Omron CX-Programmer project NewProject (CX-Programmer 9.73)

# PLC NewPLC1: CP1L M

## Global symbols (name address type ; comment)
0.00 BOOL  ; ACK
0.01 BOOL  ; RESET
0.02 BOOL  ; LAMP TEST
0.03 BOOL  ; LSH-D2017
0.04 BOOL  ; LSHH-D2017
0.05 BOOL  ; LSH-D2018
0.06 BOOL  ; LSHH-D2018
0.07 BOOL  ; LSH-O0001
0.08 BOOL  ; LSHH-O0001
0.09 BOOL  ; LSH-O0002
0.10 BOOL  ; LSHH-O0002
0.11 BOOL  ; LSH-O0003
100.00 BOOL  ; LAH-D2017
100.01 BOOL  ; LAHH-D2017
100.02 BOOL  ; LAH-D2018
100.03 BOOL  ; LAHH-D2018
100.04 BOOL  ; LAH-O0001
100.05 BOOL  ; LAHH-O0001
100.06 BOOL  ; LAH-O0002
100.07 BOOL  ; LAHH-O0002
101.00 BOOL  ; LAH-O0003
101.01 BOOL  ; LAHH-O0003
101.02 BOOL  ; LAH-O0004
101.03 BOOL  ; LAHH-O0004
101.04 BOOL  ; LAH-O0006
101.05 BOOL  ; LAHH-O0006
101.06 BOOL  ; LAH-O0008
101.07 BOOL  ; LAHH-O0008
102.00 BOOL  ; LAH-O0009
102.01 BOOL  ; LAHH-O0009
102.02 BOOL  ; LAH-O0010
102.03 BOOL  ; LAHH-O0010
102.04 BOOL  ; LAH-O0011
102.05 BOOL  ; LAHH-O0011
102.06 BOOL  ; LAH-O0012
102.07 BOOL  ; LAHH-O0012
103.00 BOOL  ; LAH-O0013
103.01 BOOL  ; LAHH-O0013
103.02 BOOL  ; LAH-O0014
103.03 BOOL  ; LAHH-O0014
103.04 BOOL  ; LAH-O0024
103.05 BOOL  ; LAHH-O0024
104.00 BOOL  ; LAH-O0025
104.01 BOOL  ; LAHH-O0025
104.02 BOOL  ; LAH-N0002
104.03 BOOL  ; LAHH-N0002
104.04 BOOL  ; LAH-N0004
104.05 BOOL  ; LAHH-N0004
104.06 BOOL  ; BUZZER
104.07 BOOL  ; HORN-LSH
105.00 BOOL  ; HORN-LSHH
105.01 BOOL  ; LIGHT-LSH
105.02 BOOL  ; LIGHT-LSHH
1.00 BOOL  ; LSHH-O0003
1.01 BOOL  ; LSH-O0004
1.02 BOOL  ; LSHH-O0004
1.03 BOOL  ; LSH-O0006
1.04 BOOL  ; LSHH-O0006
1.05 BOOL  ; LSH-O0008
1.06 BOOL  ; LSHH-O0008
2.00 BOOL  ; LSH-O0009
2.01 BOOL  ; LSHH-O0009
2.02 BOOL  ; LSH-O0010
2.03 BOOL  ; LSHH-O0010
2.04 BOOL  ; LSH-O0011
2.05 BOOL  ; LSHH-O0011
2.06 BOOL  ; LSH-O0012
2.07 BOOL  ; LSHH-O0012
2.08 BOOL  ; LSH-O0013
2.09 BOOL  ; LSHH-O0013
2.10 BOOL  ; LSH-O0014
2.11 BOOL  ; LSHH-O0014
3.00 BOOL  ; LSH-O0024
3.01 BOOL  ; LSHH-O0024
3.02 BOOL  ; LSH-O0025
3.03 BOOL  ; LSHH-O0025
3.04 BOOL  ; LSH-N0002
3.05 BOOL  ; LSHH-N0002
3.06 BOOL  ; LSH-N0004
3.07 BOOL  ; LSHH-N0004

## Program IHLAProject (cyclic task 0)

### Section RunningSystem

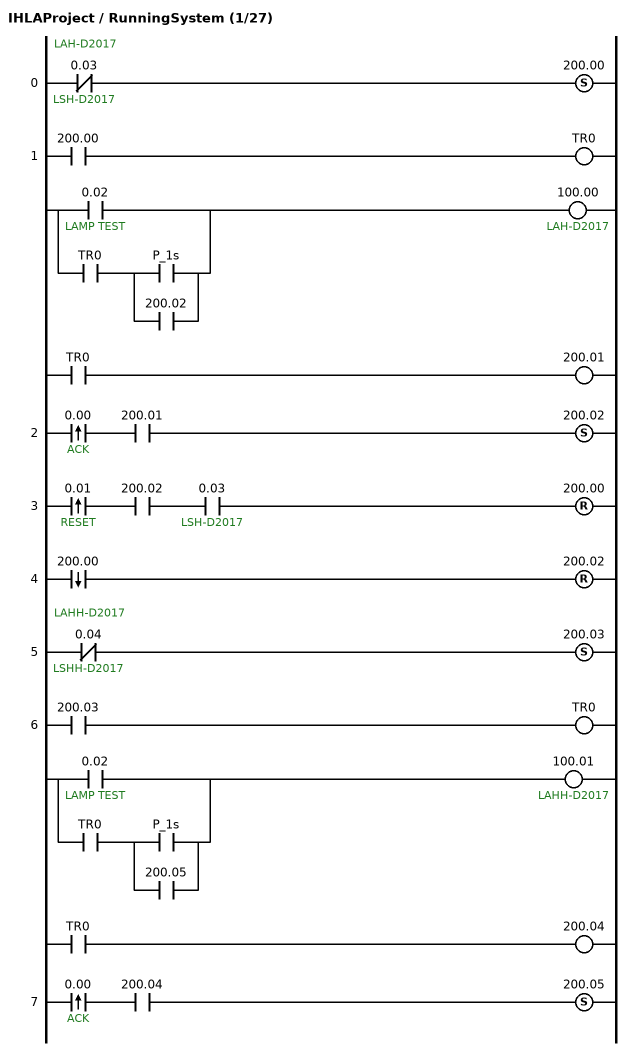
; rung 0: LAH-D2017
LDNOT 0.03  ; LSH-D2017
SET 200.00
; rung 1
LD 0.02  ; LAMP TEST
LD 200.00
OUT TR0
LD P_1s
OR 200.02
ANDLD
ORLD
OUT 100.00  ; LAH-D2017
LD TR0
OUT 200.01
; rung 2
@LD 0.00  ; ACK
AND 200.01
SET 200.02
; rung 3
@LD 0.01  ; RESET
AND 200.02
AND 0.03  ; LSH-D2017
RSET 200.00
; rung 4
%LD 200.00
RSET 200.02
; rung 5: LAHH-D2017
LDNOT 0.04  ; LSHH-D2017
SET 200.03
; rung 6
LD 0.02  ; LAMP TEST
LD 200.03
OUT TR0
LD P_1s
OR 200.05
ANDLD
ORLD
OUT 100.01  ; LAHH-D2017
LD TR0
OUT 200.04
; rung 7
@LD 0.00  ; ACK
AND 200.04
SET 200.05

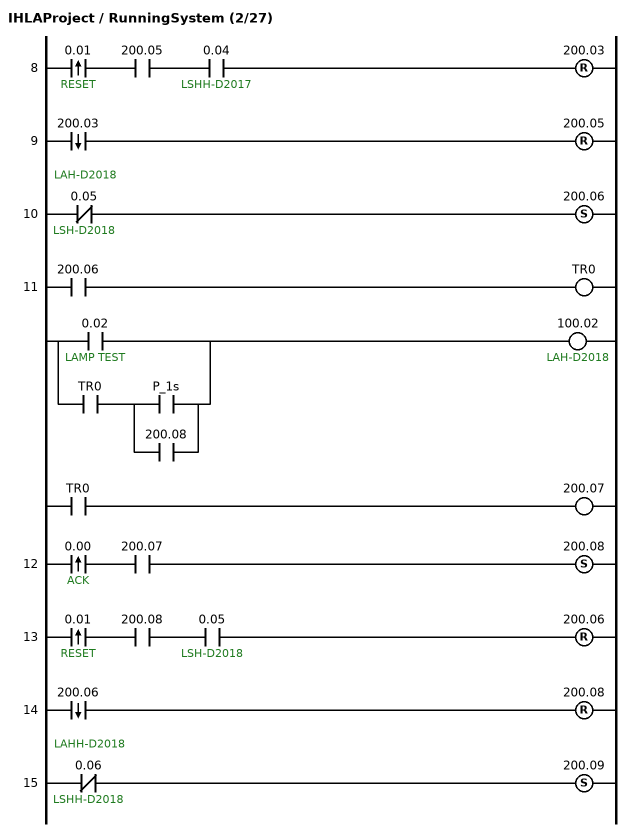
; rung 8
@LD 0.01  ; RESET
AND 200.05
AND 0.04  ; LSHH-D2017
RSET 200.03
; rung 9
%LD 200.03
RSET 200.05
; rung 10: LAH-D2018
LDNOT 0.05  ; LSH-D2018
SET 200.06
; rung 11
LD 0.02  ; LAMP TEST
LD 200.06
OUT TR0
LD P_1s
OR 200.08
ANDLD
ORLD
OUT 100.02  ; LAH-D2018
LD TR0
OUT 200.07
; rung 12
@LD 0.00  ; ACK
AND 200.07
SET 200.08
; rung 13
@LD 0.01  ; RESET
AND 200.08
AND 0.05  ; LSH-D2018
RSET 200.06
; rung 14
%LD 200.06
RSET 200.08
; rung 15: LAHH-D2018
LDNOT 0.06  ; LSHH-D2018
SET 200.09

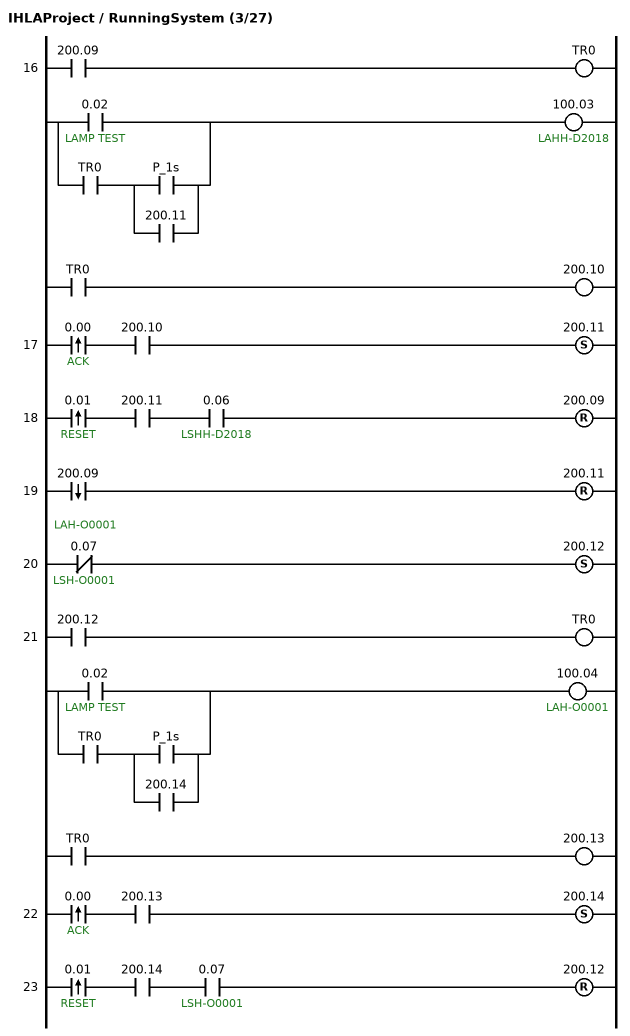
; rung 16
LD 0.02  ; LAMP TEST
LD 200.09
OUT TR0
LD P_1s
OR 200.11
ANDLD
ORLD
OUT 100.03  ; LAHH-D2018
LD TR0
OUT 200.10
; rung 17
@LD 0.00  ; ACK
AND 200.10
SET 200.11
; rung 18
@LD 0.01  ; RESET
AND 200.11
AND 0.06  ; LSHH-D2018
RSET 200.09
; rung 19
%LD 200.09
RSET 200.11
; rung 20: LAH-O0001
LDNOT 0.07  ; LSH-O0001
SET 200.12
; rung 21
LD 0.02  ; LAMP TEST
LD 200.12
OUT TR0
LD P_1s
OR 200.14
ANDLD
ORLD
OUT 100.04  ; LAH-O0001
LD TR0
OUT 200.13
; rung 22
@LD 0.00  ; ACK
AND 200.13
SET 200.14
; rung 23
@LD 0.01  ; RESET
AND 200.14
AND 0.07  ; LSH-O0001
RSET 200.12

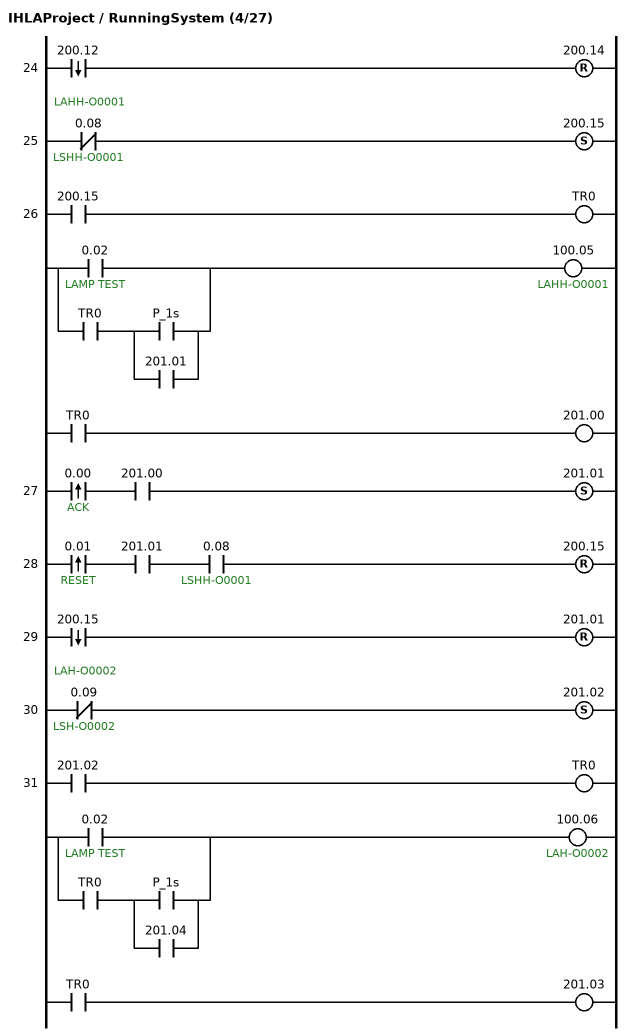
; rung 24
%LD 200.12
RSET 200.14
; rung 25: LAHH-O0001
LDNOT 0.08  ; LSHH-O0001
SET 200.15
; rung 26
LD 0.02  ; LAMP TEST
LD 200.15
OUT TR0
LD P_1s
OR 201.01
ANDLD
ORLD
OUT 100.05  ; LAHH-O0001
LD TR0
OUT 201.00
; rung 27
@LD 0.00  ; ACK
AND 201.00
SET 201.01
; rung 28
@LD 0.01  ; RESET
AND 201.01
AND 0.08  ; LSHH-O0001
RSET 200.15
; rung 29
%LD 200.15
RSET 201.01
; rung 30: LAH-O0002
LDNOT 0.09  ; LSH-O0002
SET 201.02
; rung 31
LD 0.02  ; LAMP TEST
LD 201.02
OUT TR0
LD P_1s
OR 201.04
ANDLD
ORLD
OUT 100.06  ; LAH-O0002
LD TR0
OUT 201.03

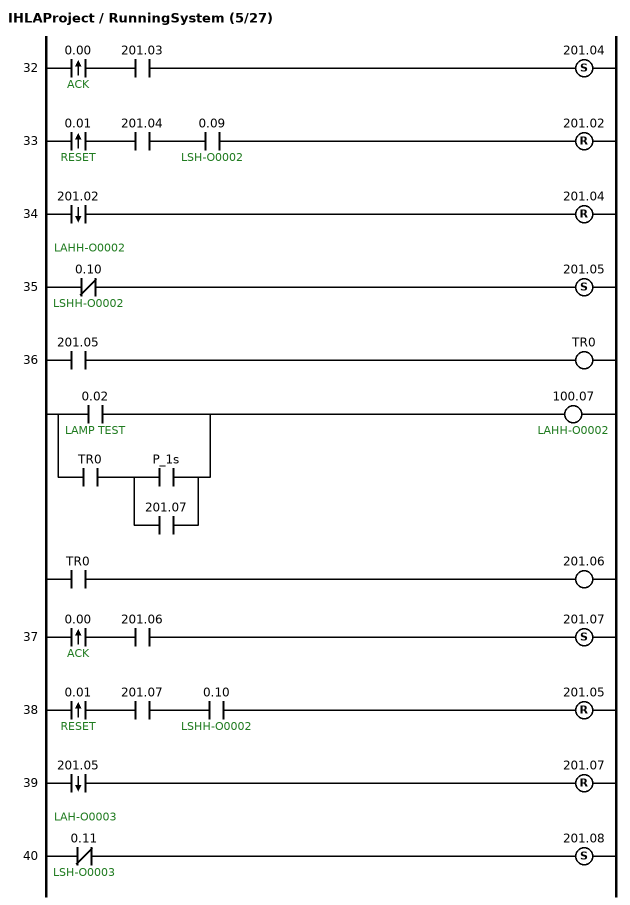
; rung 32
@LD 0.00  ; ACK
AND 201.03
SET 201.04
; rung 33
@LD 0.01  ; RESET
AND 201.04
AND 0.09  ; LSH-O0002
RSET 201.02
; rung 34
%LD 201.02
RSET 201.04
; rung 35: LAHH-O0002
LDNOT 0.10  ; LSHH-O0002
SET 201.05
; rung 36
LD 0.02  ; LAMP TEST
LD 201.05
OUT TR0
LD P_1s
OR 201.07
ANDLD
ORLD
OUT 100.07  ; LAHH-O0002
LD TR0
OUT 201.06
; rung 37
@LD 0.00  ; ACK
AND 201.06
SET 201.07
; rung 38
@LD 0.01  ; RESET
AND 201.07
AND 0.10  ; LSHH-O0002
RSET 201.05
; rung 39
%LD 201.05
RSET 201.07
; rung 40: LAH-O0003
LDNOT 0.11  ; LSH-O0003
SET 201.08

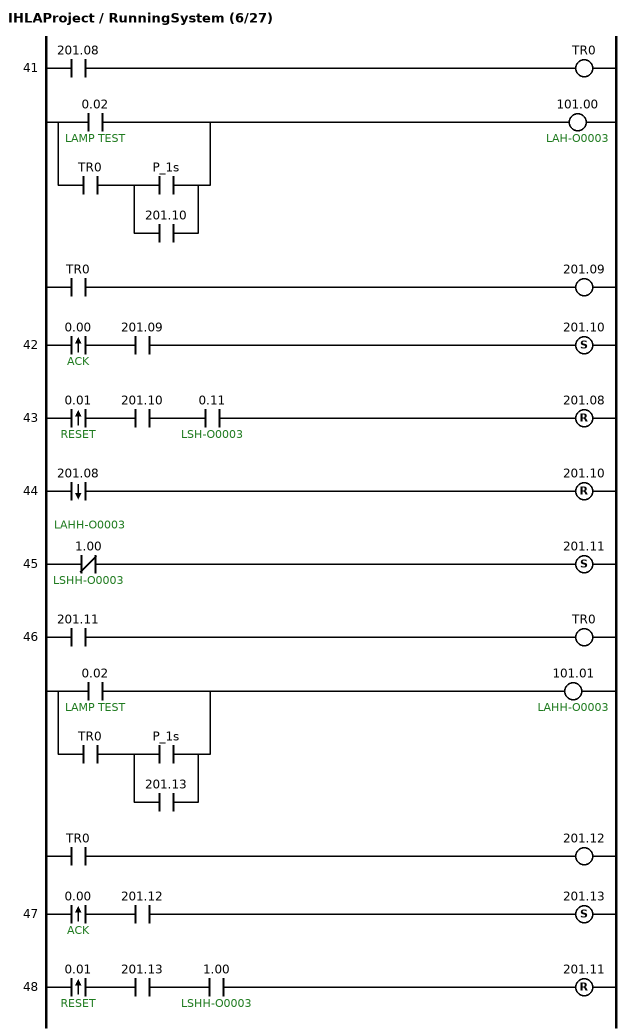
; rung 41
LD 0.02  ; LAMP TEST
LD 201.08
OUT TR0
LD P_1s
OR 201.10
ANDLD
ORLD
OUT 101.00  ; LAH-O0003
LD TR0
OUT 201.09
; rung 42
@LD 0.00  ; ACK
AND 201.09
SET 201.10
; rung 43
@LD 0.01  ; RESET
AND 201.10
AND 0.11  ; LSH-O0003
RSET 201.08
; rung 44
%LD 201.08
RSET 201.10
; rung 45: LAHH-O0003
LDNOT 1.00  ; LSHH-O0003
SET 201.11
; rung 46
LD 0.02  ; LAMP TEST
LD 201.11
OUT TR0
LD P_1s
OR 201.13
ANDLD
ORLD
OUT 101.01  ; LAHH-O0003
LD TR0
OUT 201.12
; rung 47
@LD 0.00  ; ACK
AND 201.12
SET 201.13
; rung 48
@LD 0.01  ; RESET
AND 201.13
AND 1.00  ; LSHH-O0003
RSET 201.11

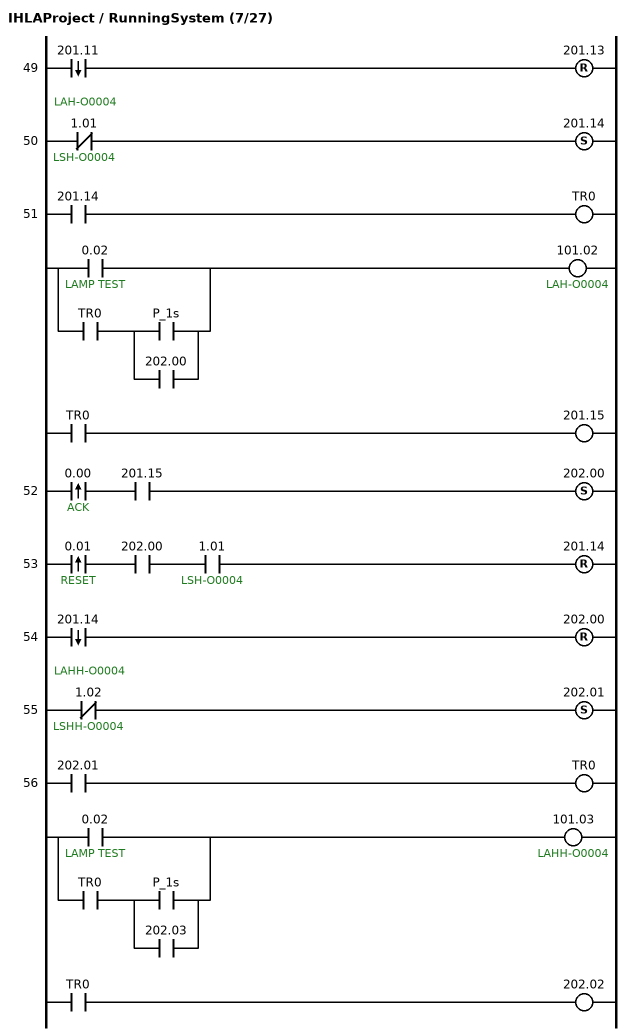
; rung 49
%LD 201.11
RSET 201.13
; rung 50: LAH-O0004
LDNOT 1.01  ; LSH-O0004
SET 201.14
; rung 51
LD 0.02  ; LAMP TEST
LD 201.14
OUT TR0
LD P_1s
OR 202.00
ANDLD
ORLD
OUT 101.02  ; LAH-O0004
LD TR0
OUT 201.15
; rung 52
@LD 0.00  ; ACK
AND 201.15
SET 202.00
; rung 53
@LD 0.01  ; RESET
AND 202.00
AND 1.01  ; LSH-O0004
RSET 201.14
; rung 54
%LD 201.14
RSET 202.00
; rung 55: LAHH-O0004
LDNOT 1.02  ; LSHH-O0004
SET 202.01
; rung 56
LD 0.02  ; LAMP TEST
LD 202.01
OUT TR0
LD P_1s
OR 202.03
ANDLD
ORLD
OUT 101.03  ; LAHH-O0004
LD TR0
OUT 202.02

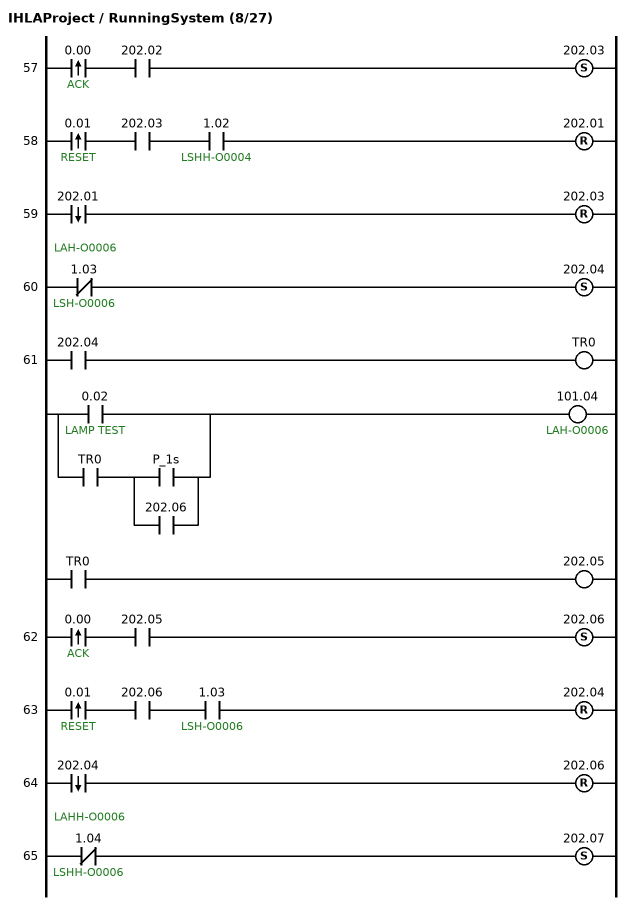
; rung 57
@LD 0.00  ; ACK
AND 202.02
SET 202.03
; rung 58
@LD 0.01  ; RESET
AND 202.03
AND 1.02  ; LSHH-O0004
RSET 202.01
; rung 59
%LD 202.01
RSET 202.03
; rung 60: LAH-O0006
LDNOT 1.03  ; LSH-O0006
SET 202.04
; rung 61
LD 0.02  ; LAMP TEST
LD 202.04
OUT TR0
LD P_1s
OR 202.06
ANDLD
ORLD
OUT 101.04  ; LAH-O0006
LD TR0
OUT 202.05
; rung 62
@LD 0.00  ; ACK
AND 202.05
SET 202.06
; rung 63
@LD 0.01  ; RESET
AND 202.06
AND 1.03  ; LSH-O0006
RSET 202.04
; rung 64
%LD 202.04
RSET 202.06
; rung 65: LAHH-O0006
LDNOT 1.04  ; LSHH-O0006
SET 202.07

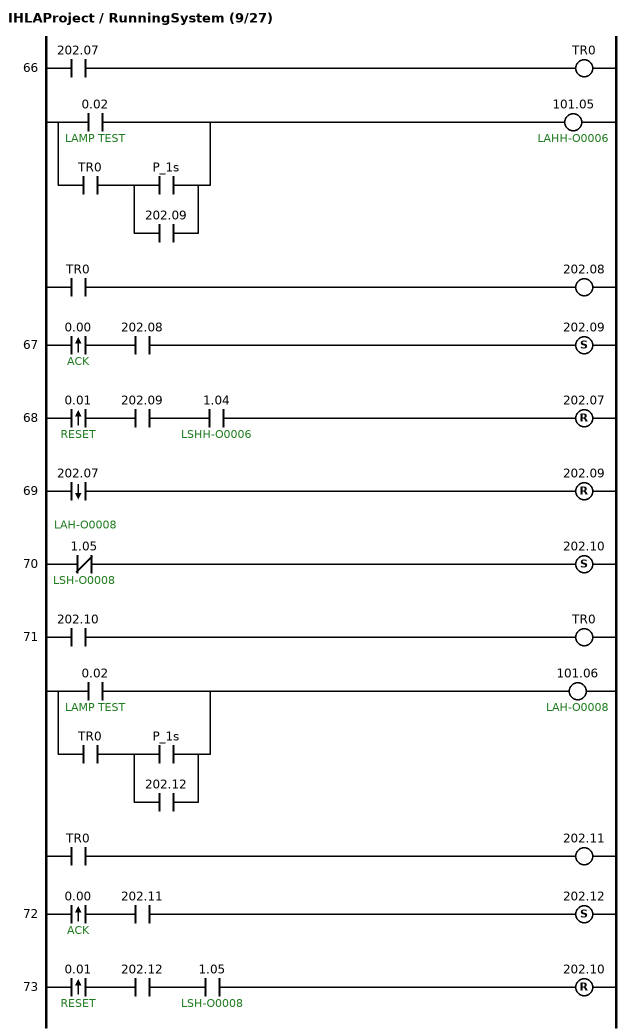
; rung 66
LD 0.02  ; LAMP TEST
LD 202.07
OUT TR0
LD P_1s
OR 202.09
ANDLD
ORLD
OUT 101.05  ; LAHH-O0006
LD TR0
OUT 202.08
; rung 67
@LD 0.00  ; ACK
AND 202.08
SET 202.09
; rung 68
@LD 0.01  ; RESET
AND 202.09
AND 1.04  ; LSHH-O0006
RSET 202.07
; rung 69
%LD 202.07
RSET 202.09
; rung 70: LAH-O0008
LDNOT 1.05  ; LSH-O0008
SET 202.10
; rung 71
LD 0.02  ; LAMP TEST
LD 202.10
OUT TR0
LD P_1s
OR 202.12
ANDLD
ORLD
OUT 101.06  ; LAH-O0008
LD TR0
OUT 202.11
; rung 72
@LD 0.00  ; ACK
AND 202.11
SET 202.12
; rung 73
@LD 0.01  ; RESET
AND 202.12
AND 1.05  ; LSH-O0008
RSET 202.10

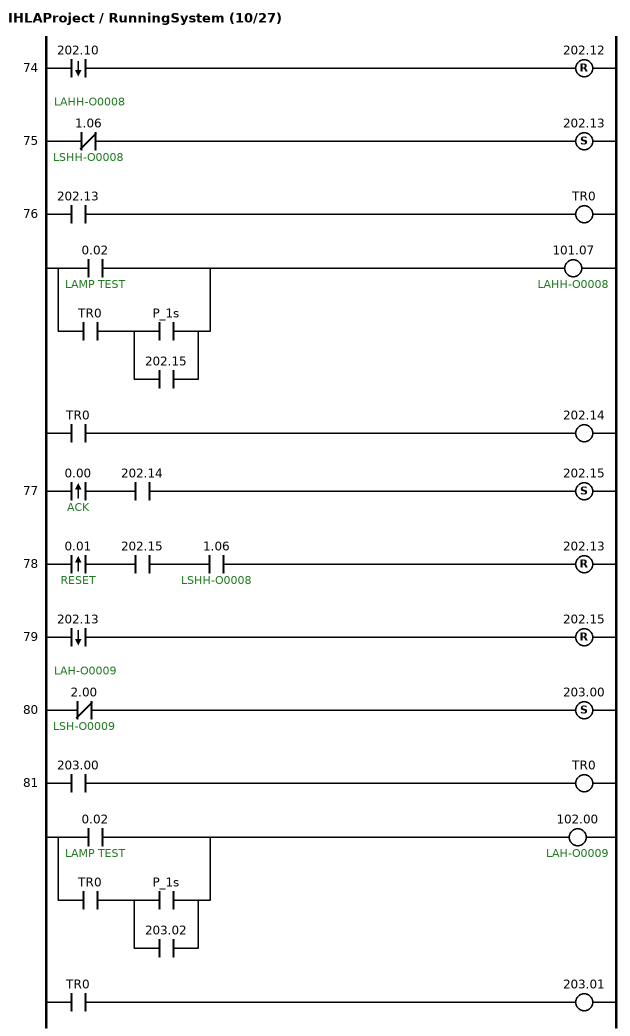
; rung 74
%LD 202.10
RSET 202.12
; rung 75: LAHH-O0008
LDNOT 1.06  ; LSHH-O0008
SET 202.13
; rung 76
LD 0.02  ; LAMP TEST
LD 202.13
OUT TR0
LD P_1s
OR 202.15
ANDLD
ORLD
OUT 101.07  ; LAHH-O0008
LD TR0
OUT 202.14
; rung 77
@LD 0.00  ; ACK
AND 202.14
SET 202.15
; rung 78
@LD 0.01  ; RESET
AND 202.15
AND 1.06  ; LSHH-O0008
RSET 202.13
; rung 79
%LD 202.13
RSET 202.15
; rung 80: LAH-O0009
LDNOT 2.00  ; LSH-O0009
SET 203.00
; rung 81
LD 0.02  ; LAMP TEST
LD 203.00
OUT TR0
LD P_1s
OR 203.02
ANDLD
ORLD
OUT 102.00  ; LAH-O0009
LD TR0
OUT 203.01

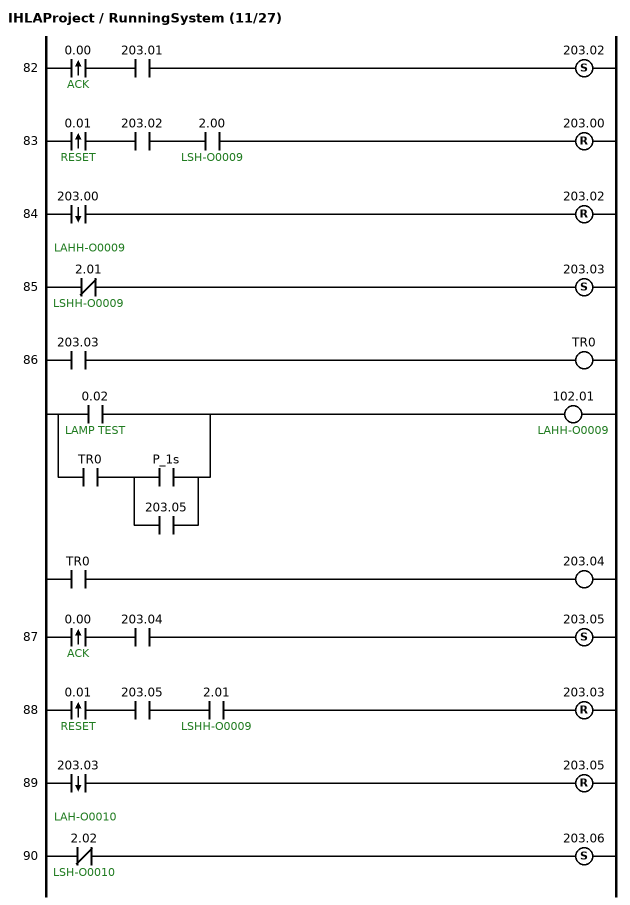
; rung 82
@LD 0.00  ; ACK
AND 203.01
SET 203.02
; rung 83
@LD 0.01  ; RESET
AND 203.02
AND 2.00  ; LSH-O0009
RSET 203.00
; rung 84
%LD 203.00
RSET 203.02
; rung 85: LAHH-O0009
LDNOT 2.01  ; LSHH-O0009
SET 203.03
; rung 86
LD 0.02  ; LAMP TEST
LD 203.03
OUT TR0
LD P_1s
OR 203.05
ANDLD
ORLD
OUT 102.01  ; LAHH-O0009
LD TR0
OUT 203.04
; rung 87
@LD 0.00  ; ACK
AND 203.04
SET 203.05
; rung 88
@LD 0.01  ; RESET
AND 203.05
AND 2.01  ; LSHH-O0009
RSET 203.03
; rung 89
%LD 203.03
RSET 203.05
; rung 90: LAH-O0010
LDNOT 2.02  ; LSH-O0010
SET 203.06

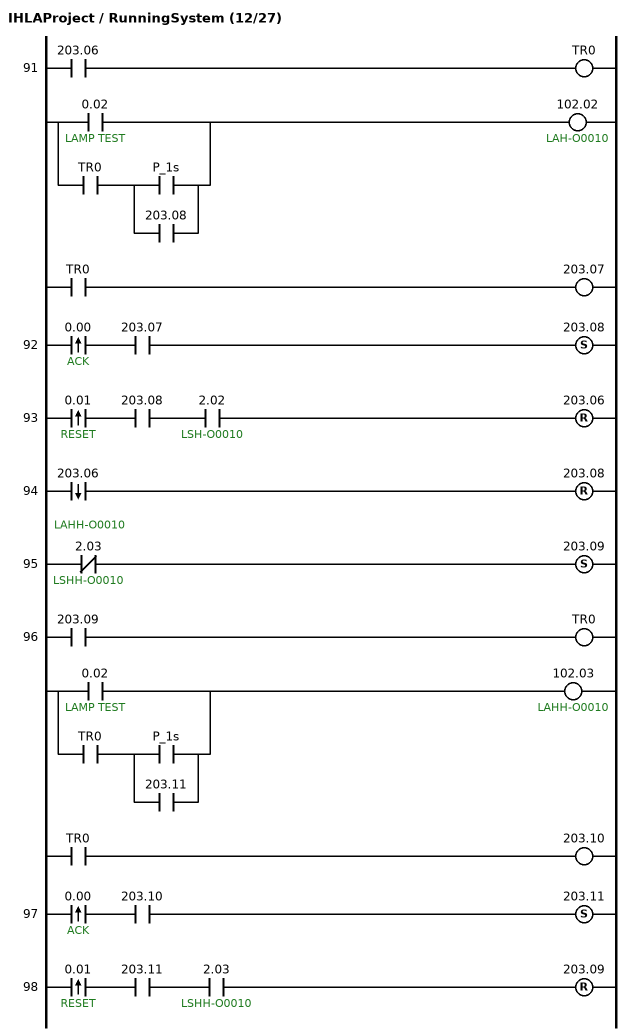
; rung 91
LD 0.02  ; LAMP TEST
LD 203.06
OUT TR0
LD P_1s
OR 203.08
ANDLD
ORLD
OUT 102.02  ; LAH-O0010
LD TR0
OUT 203.07
; rung 92
@LD 0.00  ; ACK
AND 203.07
SET 203.08
; rung 93
@LD 0.01  ; RESET
AND 203.08
AND 2.02  ; LSH-O0010
RSET 203.06
; rung 94
%LD 203.06
RSET 203.08
; rung 95: LAHH-O0010
LDNOT 2.03  ; LSHH-O0010
SET 203.09
; rung 96
LD 0.02  ; LAMP TEST
LD 203.09
OUT TR0
LD P_1s
OR 203.11
ANDLD
ORLD
OUT 102.03  ; LAHH-O0010
LD TR0
OUT 203.10
; rung 97
@LD 0.00  ; ACK
AND 203.10
SET 203.11
; rung 98
@LD 0.01  ; RESET
AND 203.11
AND 2.03  ; LSHH-O0010
RSET 203.09

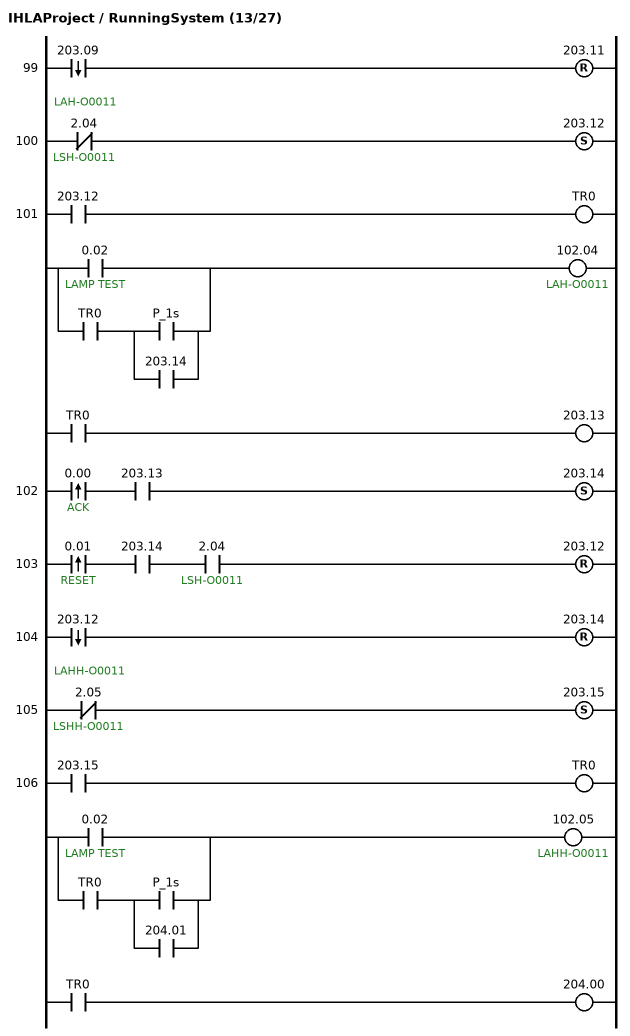
; rung 99
%LD 203.09
RSET 203.11
; rung 100: LAH-O0011
LDNOT 2.04  ; LSH-O0011
SET 203.12
; rung 101
LD 0.02  ; LAMP TEST
LD 203.12
OUT TR0
LD P_1s
OR 203.14
ANDLD
ORLD
OUT 102.04  ; LAH-O0011
LD TR0
OUT 203.13
; rung 102
@LD 0.00  ; ACK
AND 203.13
SET 203.14
; rung 103
@LD 0.01  ; RESET
AND 203.14
AND 2.04  ; LSH-O0011
RSET 203.12
; rung 104
%LD 203.12
RSET 203.14
; rung 105: LAHH-O0011
LDNOT 2.05  ; LSHH-O0011
SET 203.15
; rung 106
LD 0.02  ; LAMP TEST
LD 203.15
OUT TR0
LD P_1s
OR 204.01
ANDLD
ORLD
OUT 102.05  ; LAHH-O0011
LD TR0
OUT 204.00

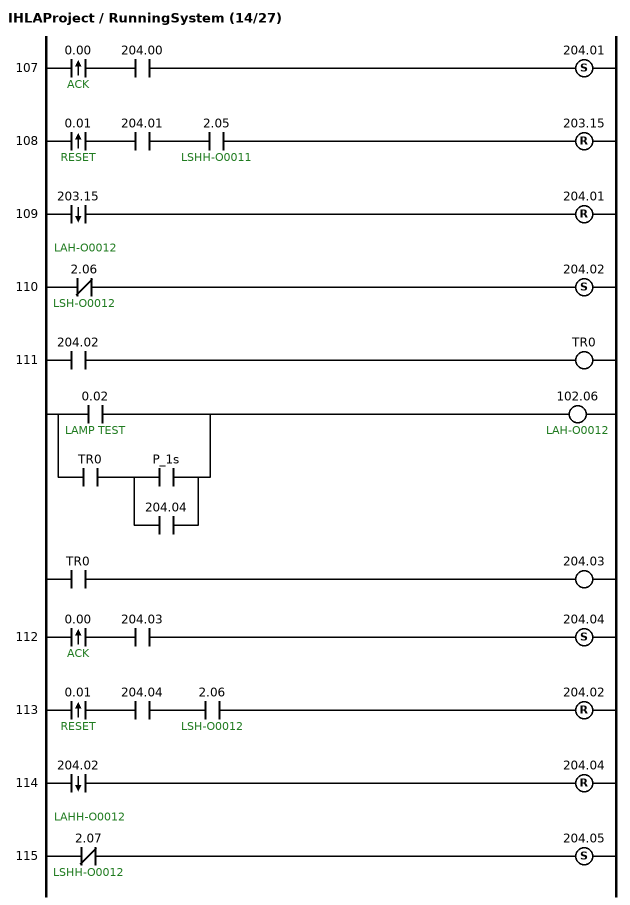
; rung 107
@LD 0.00  ; ACK
AND 204.00
SET 204.01
; rung 108
@LD 0.01  ; RESET
AND 204.01
AND 2.05  ; LSHH-O0011
RSET 203.15
; rung 109
%LD 203.15
RSET 204.01
; rung 110: LAH-O0012
LDNOT 2.06  ; LSH-O0012
SET 204.02
; rung 111
LD 0.02  ; LAMP TEST
LD 204.02
OUT TR0
LD P_1s
OR 204.04
ANDLD
ORLD
OUT 102.06  ; LAH-O0012
LD TR0
OUT 204.03
; rung 112
@LD 0.00  ; ACK
AND 204.03
SET 204.04
; rung 113
@LD 0.01  ; RESET
AND 204.04
AND 2.06  ; LSH-O0012
RSET 204.02
; rung 114
%LD 204.02
RSET 204.04
; rung 115: LAHH-O0012
LDNOT 2.07  ; LSHH-O0012
SET 204.05

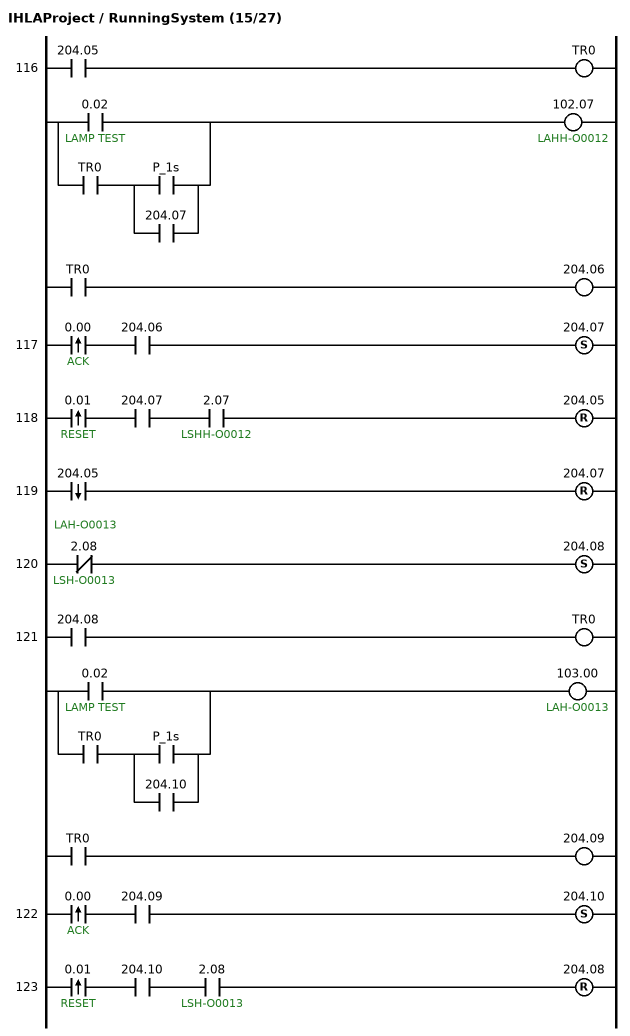
; rung 116
LD 0.02  ; LAMP TEST
LD 204.05
OUT TR0
LD P_1s
OR 204.07
ANDLD
ORLD
OUT 102.07  ; LAHH-O0012
LD TR0
OUT 204.06
; rung 117
@LD 0.00  ; ACK
AND 204.06
SET 204.07
; rung 118
@LD 0.01  ; RESET
AND 204.07
AND 2.07  ; LSHH-O0012
RSET 204.05
; rung 119
%LD 204.05
RSET 204.07
; rung 120: LAH-O0013
LDNOT 2.08  ; LSH-O0013
SET 204.08
; rung 121
LD 0.02  ; LAMP TEST
LD 204.08
OUT TR0
LD P_1s
OR 204.10
ANDLD
ORLD
OUT 103.00  ; LAH-O0013
LD TR0
OUT 204.09
; rung 122
@LD 0.00  ; ACK
AND 204.09
SET 204.10
; rung 123
@LD 0.01  ; RESET
AND 204.10
AND 2.08  ; LSH-O0013
RSET 204.08

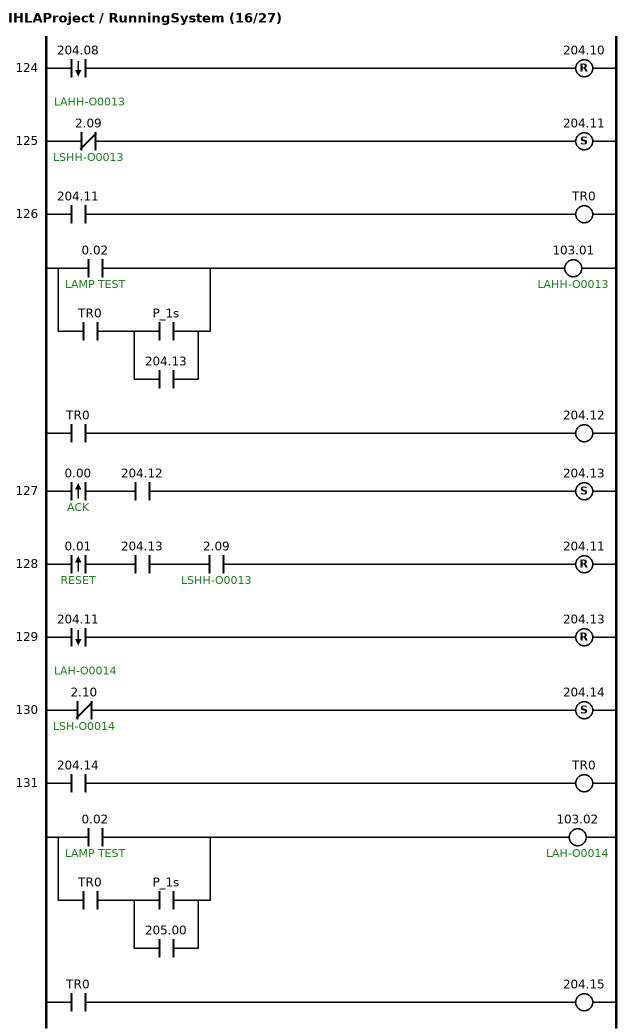
; rung 124
%LD 204.08
RSET 204.10
; rung 125: LAHH-O0013
LDNOT 2.09  ; LSHH-O0013
SET 204.11
; rung 126
LD 0.02  ; LAMP TEST
LD 204.11
OUT TR0
LD P_1s
OR 204.13
ANDLD
ORLD
OUT 103.01  ; LAHH-O0013
LD TR0
OUT 204.12
; rung 127
@LD 0.00  ; ACK
AND 204.12
SET 204.13
; rung 128
@LD 0.01  ; RESET
AND 204.13
AND 2.09  ; LSHH-O0013
RSET 204.11
; rung 129
%LD 204.11
RSET 204.13
; rung 130: LAH-O0014
LDNOT 2.10  ; LSH-O0014
SET 204.14
; rung 131
LD 0.02  ; LAMP TEST
LD 204.14
OUT TR0
LD P_1s
OR 205.00
ANDLD
ORLD
OUT 103.02  ; LAH-O0014
LD TR0
OUT 204.15

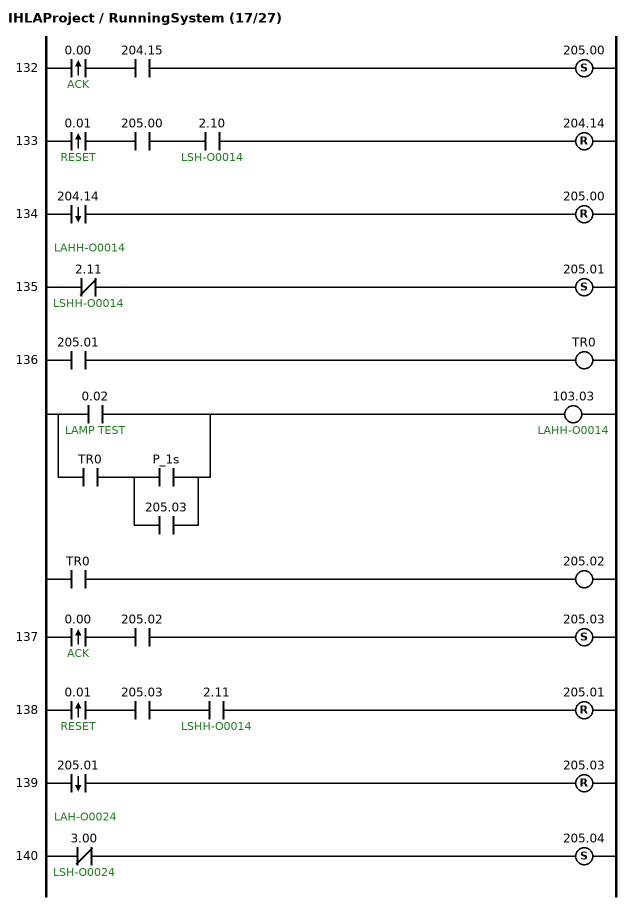
; rung 132
@LD 0.00  ; ACK
AND 204.15
SET 205.00
; rung 133
@LD 0.01  ; RESET
AND 205.00
AND 2.10  ; LSH-O0014
RSET 204.14
; rung 134
%LD 204.14
RSET 205.00
; rung 135: LAHH-O0014
LDNOT 2.11  ; LSHH-O0014
SET 205.01
; rung 136
LD 0.02  ; LAMP TEST
LD 205.01
OUT TR0
LD P_1s
OR 205.03
ANDLD
ORLD
OUT 103.03  ; LAHH-O0014
LD TR0
OUT 205.02
; rung 137
@LD 0.00  ; ACK
AND 205.02
SET 205.03
; rung 138
@LD 0.01  ; RESET
AND 205.03
AND 2.11  ; LSHH-O0014
RSET 205.01
; rung 139
%LD 205.01
RSET 205.03
; rung 140: LAH-O0024
LDNOT 3.00  ; LSH-O0024
SET 205.04

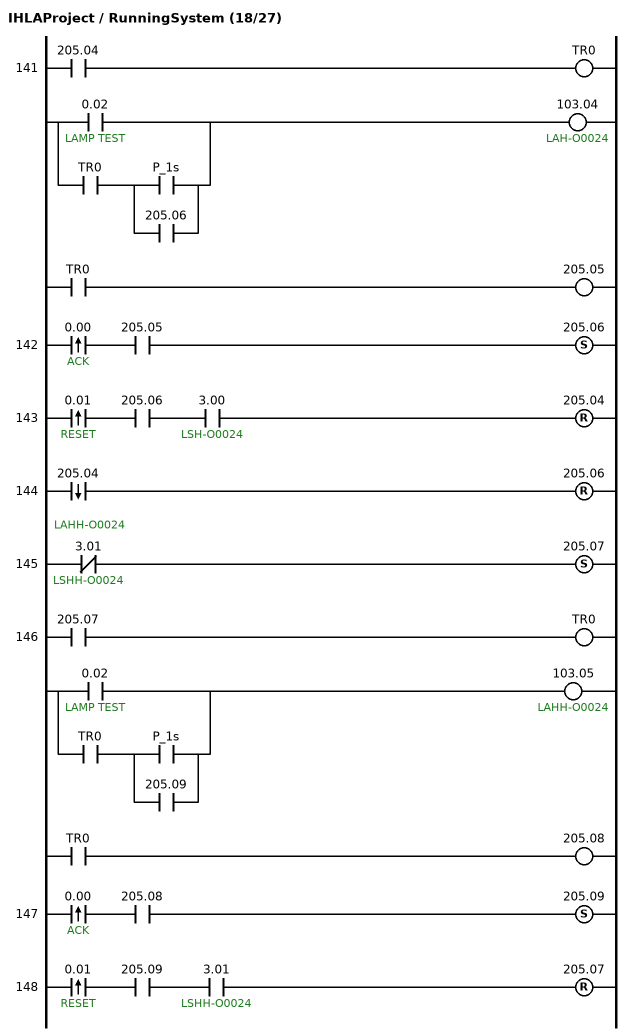
; rung 141
LD 0.02  ; LAMP TEST
LD 205.04
OUT TR0
LD P_1s
OR 205.06
ANDLD
ORLD
OUT 103.04  ; LAH-O0024
LD TR0
OUT 205.05
; rung 142
@LD 0.00  ; ACK
AND 205.05
SET 205.06
; rung 143
@LD 0.01  ; RESET
AND 205.06
AND 3.00  ; LSH-O0024
RSET 205.04
; rung 144
%LD 205.04
RSET 205.06
; rung 145: LAHH-O0024
LDNOT 3.01  ; LSHH-O0024
SET 205.07
; rung 146
LD 0.02  ; LAMP TEST
LD 205.07
OUT TR0
LD P_1s
OR 205.09
ANDLD
ORLD
OUT 103.05  ; LAHH-O0024
LD TR0
OUT 205.08
; rung 147
@LD 0.00  ; ACK
AND 205.08
SET 205.09
; rung 148
@LD 0.01  ; RESET
AND 205.09
AND 3.01  ; LSHH-O0024
RSET 205.07

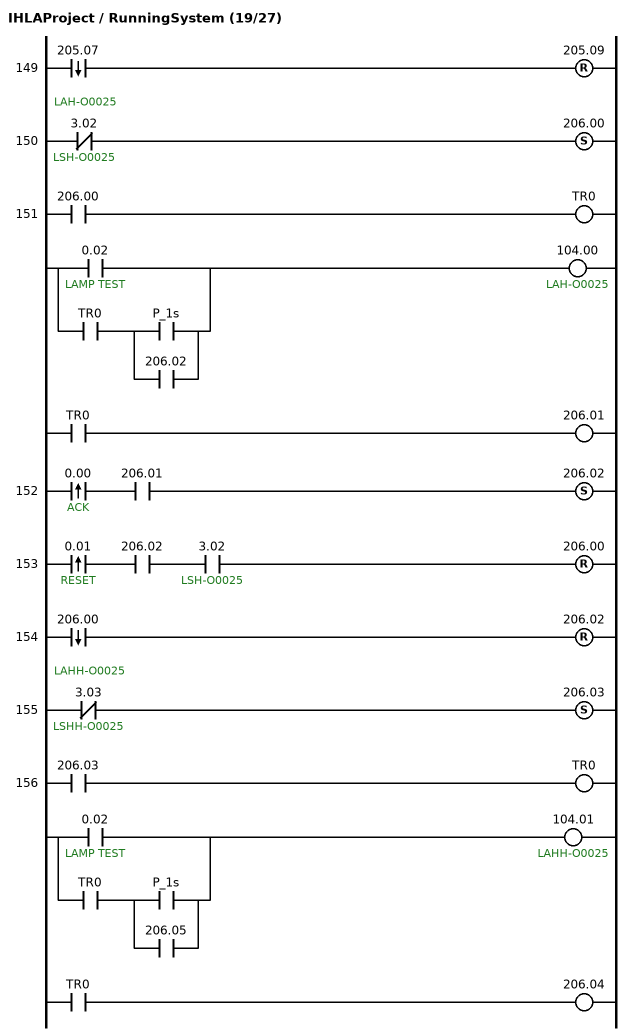
; rung 149
%LD 205.07
RSET 205.09
; rung 150: LAH-O0025
LDNOT 3.02  ; LSH-O0025
SET 206.00
; rung 151
LD 0.02  ; LAMP TEST
LD 206.00
OUT TR0
LD P_1s
OR 206.02
ANDLD
ORLD
OUT 104.00  ; LAH-O0025
LD TR0
OUT 206.01
; rung 152
@LD 0.00  ; ACK
AND 206.01
SET 206.02
; rung 153
@LD 0.01  ; RESET
AND 206.02
AND 3.02  ; LSH-O0025
RSET 206.00
; rung 154
%LD 206.00
RSET 206.02
; rung 155: LAHH-O0025
LDNOT 3.03  ; LSHH-O0025
SET 206.03
; rung 156
LD 0.02  ; LAMP TEST
LD 206.03
OUT TR0
LD P_1s
OR 206.05
ANDLD
ORLD
OUT 104.01  ; LAHH-O0025
LD TR0
OUT 206.04

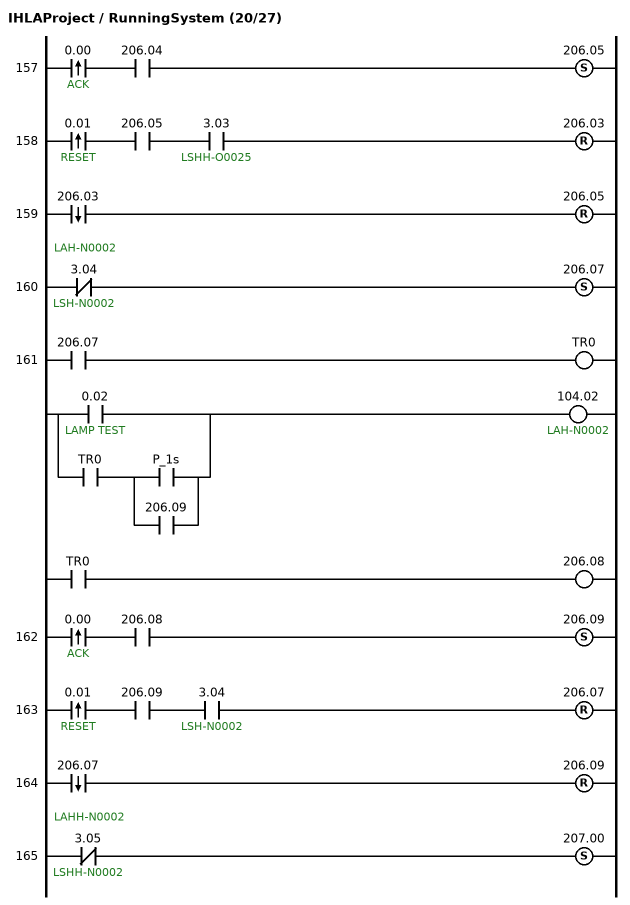
; rung 157
@LD 0.00  ; ACK
AND 206.04
SET 206.05
; rung 158
@LD 0.01  ; RESET
AND 206.05
AND 3.03  ; LSHH-O0025
RSET 206.03
; rung 159
%LD 206.03
RSET 206.05
; rung 160: LAH-N0002
LDNOT 3.04  ; LSH-N0002
SET 206.07
; rung 161
LD 0.02  ; LAMP TEST
LD 206.07
OUT TR0
LD P_1s
OR 206.09
ANDLD
ORLD
OUT 104.02  ; LAH-N0002
LD TR0
OUT 206.08
; rung 162
@LD 0.00  ; ACK
AND 206.08
SET 206.09
; rung 163
@LD 0.01  ; RESET
AND 206.09
AND 3.04  ; LSH-N0002
RSET 206.07
; rung 164
%LD 206.07
RSET 206.09
; rung 165: LAHH-N0002
LDNOT 3.05  ; LSHH-N0002
SET 207.00

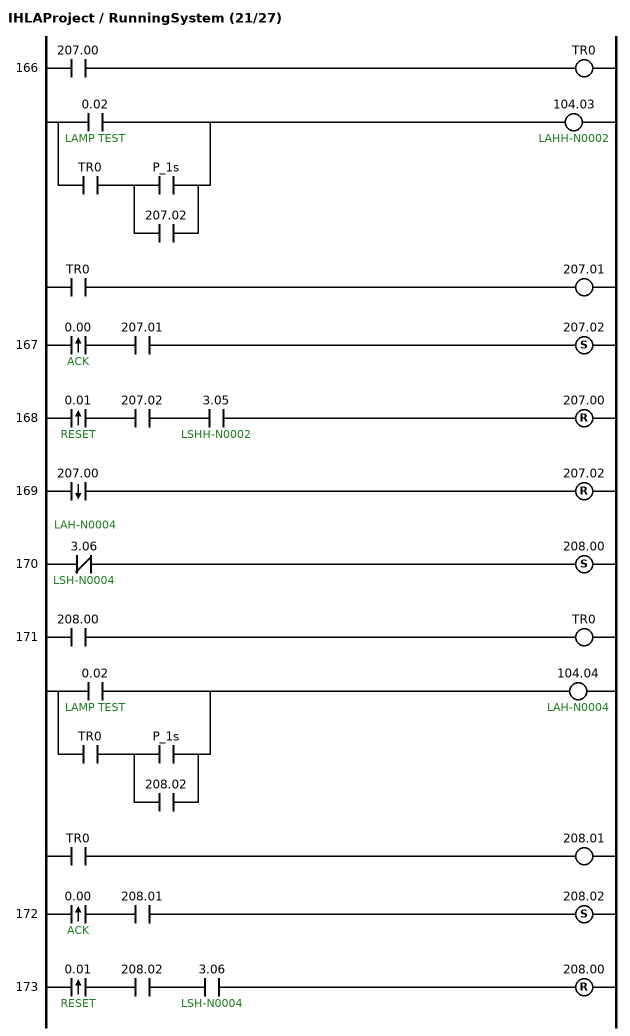
; rung 166
LD 0.02  ; LAMP TEST
LD 207.00
OUT TR0
LD P_1s
OR 207.02
ANDLD
ORLD
OUT 104.03  ; LAHH-N0002
LD TR0
OUT 207.01
; rung 167
@LD 0.00  ; ACK
AND 207.01
SET 207.02
; rung 168
@LD 0.01  ; RESET
AND 207.02
AND 3.05  ; LSHH-N0002
RSET 207.00
; rung 169
%LD 207.00
RSET 207.02
; rung 170: LAH-N0004
LDNOT 3.06  ; LSH-N0004
SET 208.00
; rung 171
LD 0.02  ; LAMP TEST
LD 208.00
OUT TR0
LD P_1s
OR 208.02
ANDLD
ORLD
OUT 104.04  ; LAH-N0004
LD TR0
OUT 208.01
; rung 172
@LD 0.00  ; ACK
AND 208.01
SET 208.02
; rung 173
@LD 0.01  ; RESET
AND 208.02
AND 3.06  ; LSH-N0004
RSET 208.00

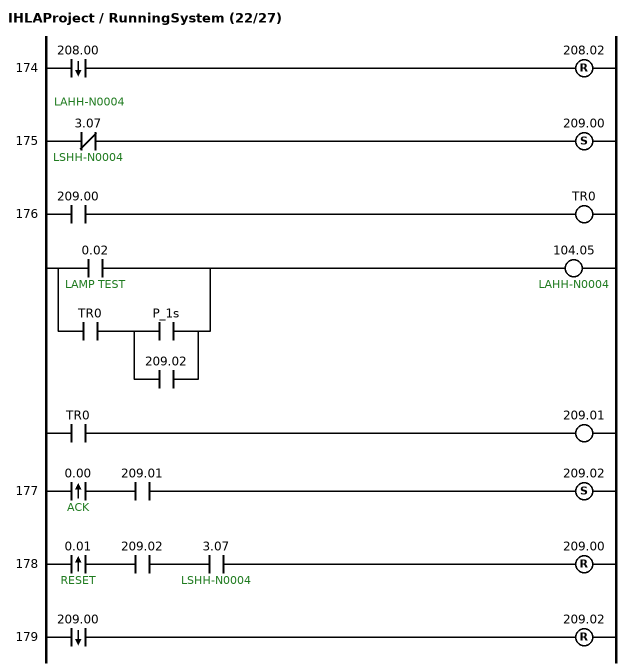
; rung 174
%LD 208.00
RSET 208.02
; rung 175: LAHH-N0004
LDNOT 3.07  ; LSHH-N0004
SET 209.00
; rung 176
LD 0.02  ; LAMP TEST
LD 209.00
OUT TR0
LD P_1s
OR 209.02
ANDLD
ORLD
OUT 104.05  ; LAHH-N0004
LD TR0
OUT 209.01
; rung 177
@LD 0.00  ; ACK
AND 209.01
SET 209.02
; rung 178
@LD 0.01  ; RESET
AND 209.02
AND 3.07  ; LSHH-N0004
RSET 209.00
; rung 179
%LD 209.00
RSET 209.02

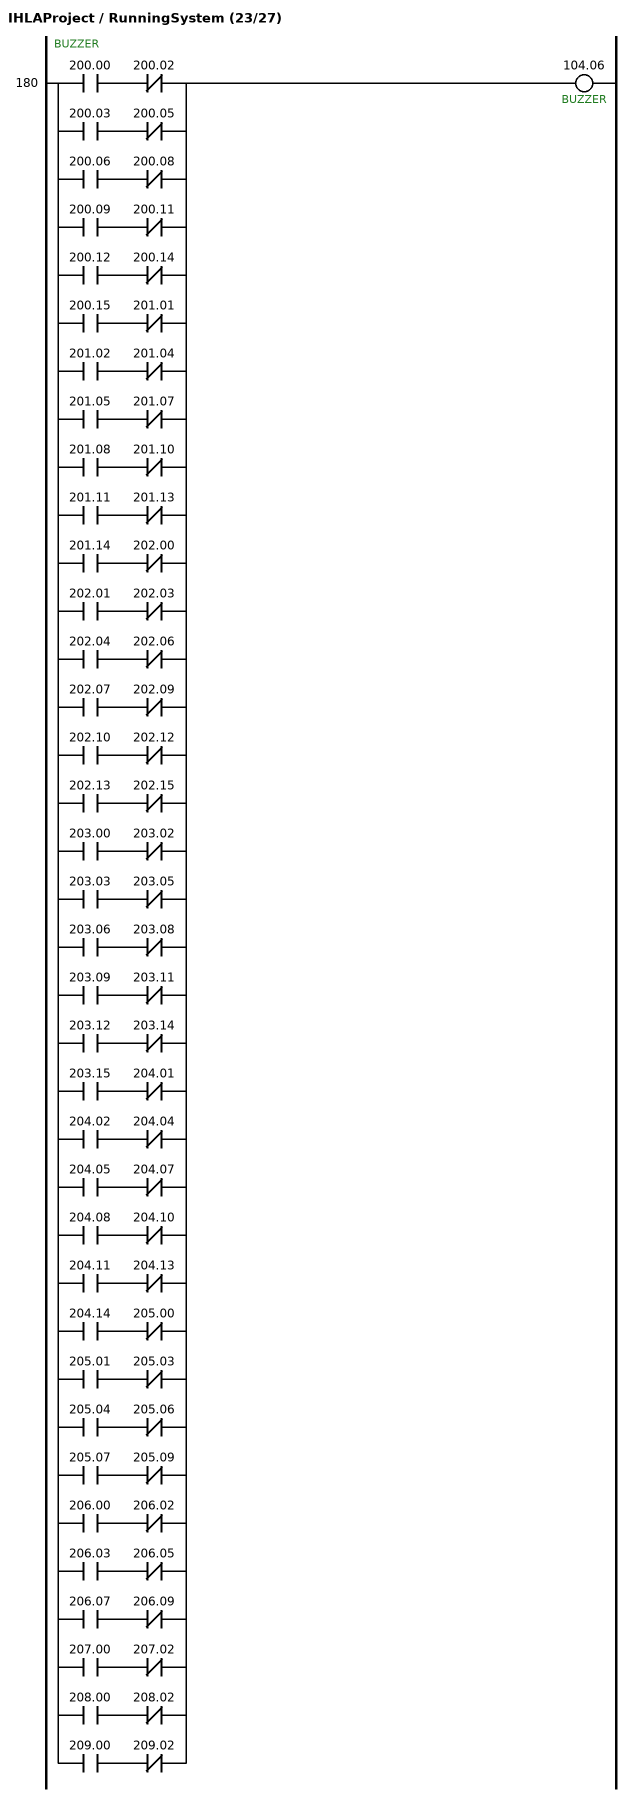
; rung 180: BUZZER
LD 200.00
ANDNOT 200.02
LD 200.03
ANDNOT 200.05
ORLD
LD 200.06
ANDNOT 200.08
ORLD
LD 200.09
ANDNOT 200.11
ORLD
LD 200.12
ANDNOT 200.14
ORLD
LD 200.15
ANDNOT 201.01
ORLD
LD 201.02
ANDNOT 201.04
ORLD
LD 201.05
ANDNOT 201.07
ORLD
LD 201.08
ANDNOT 201.10
ORLD
LD 201.11
ANDNOT 201.13
ORLD
LD 201.14
ANDNOT 202.00
ORLD
LD 202.01
ANDNOT 202.03
ORLD
LD 202.04
ANDNOT 202.06
ORLD
LD 202.07
ANDNOT 202.09
ORLD
LD 202.10
ANDNOT 202.12
ORLD
LD 202.13
ANDNOT 202.15
ORLD
LD 203.00
ANDNOT 203.02
ORLD
LD 203.03
ANDNOT 203.05
ORLD
LD 203.06
ANDNOT 203.08
ORLD
LD 203.09
ANDNOT 203.11
ORLD
LD 203.12
ANDNOT 203.14
ORLD
LD 203.15
ANDNOT 204.01
ORLD
LD 204.02
ANDNOT 204.04
ORLD
LD 204.05
ANDNOT 204.07
ORLD
LD 204.08
ANDNOT 204.10
ORLD
LD 204.11
ANDNOT 204.13
ORLD
LD 204.14
ANDNOT 205.00
ORLD
LD 205.01
ANDNOT 205.03
ORLD
LD 205.04
ANDNOT 205.06
ORLD
LD 205.07
ANDNOT 205.09
ORLD
LD 206.00
ANDNOT 206.02
ORLD
LD 206.03
ANDNOT 206.05
ORLD
LD 206.07
ANDNOT 206.09
ORLD
LD 207.00
ANDNOT 207.02
ORLD
LD 208.00
ANDNOT 208.02
ORLD
LD 209.00
ANDNOT 209.02
ORLD
OUT 104.06  ; BUZZER

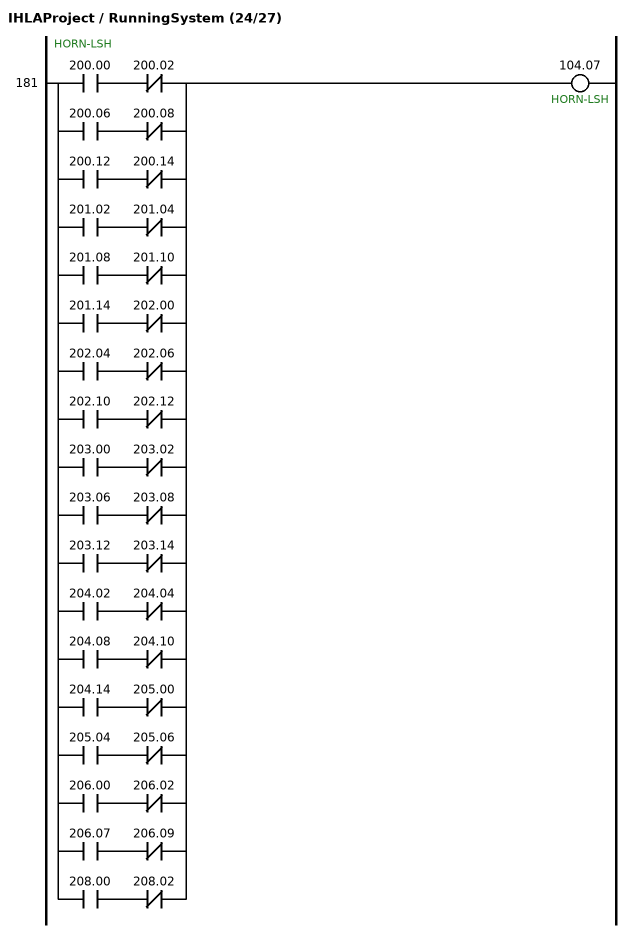
; rung 181: HORN-LSH
LD 200.00
ANDNOT 200.02
LD 200.06
ANDNOT 200.08
ORLD
LD 200.12
ANDNOT 200.14
ORLD
LD 201.02
ANDNOT 201.04
ORLD
LD 201.08
ANDNOT 201.10
ORLD
LD 201.14
ANDNOT 202.00
ORLD
LD 202.04
ANDNOT 202.06
ORLD
LD 202.10
ANDNOT 202.12
ORLD
LD 203.00
ANDNOT 203.02
ORLD
LD 203.06
ANDNOT 203.08
ORLD
LD 203.12
ANDNOT 203.14
ORLD
LD 204.02
ANDNOT 204.04
ORLD
LD 204.08
ANDNOT 204.10
ORLD
LD 204.14
ANDNOT 205.00
ORLD
LD 205.04
ANDNOT 205.06
ORLD
LD 206.00
ANDNOT 206.02
ORLD
LD 206.07
ANDNOT 206.09
ORLD
LD 208.00
ANDNOT 208.02
ORLD
OUT 104.07  ; HORN-LSH

